(* IEC 61131-3 sources: Multi-PLC-Water-Treatment-Testbed/, 3 files *)

(* ---- plc1_intake.st ---- *)
(* =========================================================================
   PLC1 - INTAKE
   Multi-PLC Water Treatment Testbed
   ---------------------------------------------------------------------------
   Raw-water source intake. Controls the intake pump that fills the treatment
   feed tank, with self-contained process simulation.

   OpenPLC / MatIEC gotchas encoded below:
     1. Located vars (AT %...) and non-located helpers MUST be in SEPARATE
        VAR blocks, else "invalid located variable declaration".
     2. OpenPLC IGNORES initial values on located vars (I/O memory is zeroed
        at start-up). Initialise them in the body on the first scan instead,
        gated by a NON-located first_scan flag (non-located inits ARE honoured).

   Modbus: %MWn -> Holding Register n; %QXn -> Coil. See docs/modbus-map.md.
   ========================================================================= *)

PROGRAM prog0
  VAR
    (* --- Located variables (Modbus-exposed) - NO initial values here --- *)
    source_level     AT %MW0  : INT;
    tank_level       AT %MW1  : INT;
    intake_flow      AT %MW2  : INT;
    pump_status      AT %MW3  : INT;
    pump_cmd         AT %QX0.0 : BOOL;
    low_source_alarm AT %QX0.1 : BOOL;
    tank_high_alarm  AT %QX0.2 : BOOL;
  END_VAR

  VAR
    (* --- Non-located helpers (separate block; inits honoured) --- *)
    first_scan : BOOL := TRUE;
    tick       : INT := 0;
  END_VAR

  (* First-scan initialisation - the only reliable way to seed located vars *)
  IF first_scan THEN
    source_level := 800;
    tank_level   := 300;
    pump_cmd     := TRUE;
    first_scan   := FALSE;
  END_IF;

  tick := tick + 1;
  IF tick >= 20 THEN          (* update process model ~1 Hz at 50 ms scan *)
    tick := 0;

    (* Dry-run protection *)
    IF source_level < 50 THEN
      low_source_alarm := TRUE;
    ELSE
      low_source_alarm := FALSE;
    END_IF;

    (* Pump moves water from source to feed tank when commanded and safe *)
    IF pump_cmd AND (source_level >= 50) THEN
      intake_flow := 100;
      pump_status := 1;
      IF source_level > 0 THEN source_level := source_level - 1; END_IF;
      IF tank_level < 1000 THEN tank_level := tank_level + 2; END_IF;
    ELSE
      intake_flow := 0;
      pump_status := 0;
    END_IF;

    (* Feed tank drains downstream *)
    IF tank_level > 0 THEN tank_level := tank_level - 1; END_IF;

    (* Overflow alarm *)
    IF tank_level >= 950 THEN
      tank_high_alarm := TRUE;
    ELSE
      tank_high_alarm := FALSE;
    END_IF;
  END_IF;
END_PROGRAM

CONFIGURATION Config0
  RESOURCE Res0 ON PLC
    TASK task0(INTERVAL := T#50ms, PRIORITY := 0);
    PROGRAM instance0 WITH task0 : prog0;
  END_RESOURCE
END_CONFIGURATION

(* ---- plc2_treatment.st ---- *)
(* =========================================================================
   PLC2 - TREATMENT
   Multi-PLC Water Treatment Testbed
   ---------------------------------------------------------------------------
   Safety-critical stage: chlorine residual dosing and pH correction.
   Headline attack: zeroing chlorine_setpoint drives chlorine to 0 and raises
   unsafe_water_alarm.

   Scaling: chlorine/pH in hundredths (200 = 2.00 mg/L, 700 = pH 7.00).
   Safe chlorine residual >= 0.50 mg/L (value >= 50).

   OpenPLC gotchas: located vs non-located in SEPARATE VAR blocks; located
   initial values are ignored at runtime, so seed them on first scan.
   See docs/modbus-map.md.
   ========================================================================= *)

PROGRAM prog0
  VAR
    (* --- Located variables (Modbus-exposed) - NO initial values here --- *)
    chlorine_level     AT %MW0  : INT;
    chlorine_setpoint  AT %MW1  : INT;
    ph_level           AT %MW2  : INT;
    ph_setpoint        AT %MW3  : INT;
    dosing_status      AT %MW4  : INT;
    dosing_enable      AT %QX0.0 : BOOL;
    unsafe_water_alarm AT %QX0.1 : BOOL;
    ph_excursion_alarm AT %QX0.2 : BOOL;
  END_VAR

  VAR
    first_scan : BOOL := TRUE;
    tick       : INT := 0;
  END_VAR

  IF first_scan THEN
    chlorine_level    := 200;
    chlorine_setpoint := 200;
    ph_level          := 700;
    ph_setpoint       := 700;
    dosing_status     := 1;
    dosing_enable     := TRUE;
    first_scan        := FALSE;
  END_IF;

  tick := tick + 1;
  IF tick >= 20 THEN
    tick := 0;

    (* Chlorine trends toward setpoint while dosing enabled; setpoint 0 -> decay *)
    IF dosing_enable THEN
      dosing_status := 1;
      IF chlorine_level < chlorine_setpoint THEN
        chlorine_level := chlorine_level + 5;
      ELSIF chlorine_level > chlorine_setpoint THEN
        chlorine_level := chlorine_level - 5;
      END_IF;
    ELSE
      dosing_status := 0;
      IF chlorine_level > 0 THEN chlorine_level := chlorine_level - 5; END_IF;
    END_IF;
    IF chlorine_level < 0 THEN chlorine_level := 0; END_IF;

    (* pH correction trends toward setpoint *)
    IF ph_level < ph_setpoint THEN
      ph_level := ph_level + 2;
    ELSIF ph_level > ph_setpoint THEN
      ph_level := ph_level - 2;
    END_IF;

    (* Safety invariants *)
    IF chlorine_level < 50 THEN
      unsafe_water_alarm := TRUE;
    ELSE
      unsafe_water_alarm := FALSE;
    END_IF;

    IF (ph_level < 650) OR (ph_level > 850) THEN
      ph_excursion_alarm := TRUE;
    ELSE
      ph_excursion_alarm := FALSE;
    END_IF;
  END_IF;
END_PROGRAM

CONFIGURATION Config0
  RESOURCE Res0 ON PLC
    TASK task0(INTERVAL := T#50ms, PRIORITY := 0);
    PROGRAM instance0 WITH task0 : prog0;
  END_RESOURCE
END_CONFIGURATION

(* ---- plc3_distribution.st ---- *)
(* =========================================================================
   PLC3 - DISTRIBUTION
   Multi-PLC Water Treatment Testbed
   ---------------------------------------------------------------------------
   Pressure management and supply via two booster pumps with a pressure-relief
   limit. Attacks: (a) pumps forced OFF -> supply failure; (b) pressure_max
   raised -> relief disabled -> overpressure.

   Scaling: pressure in hundredths of bar (800 = 8.00 bar). Safe hard limit
   = 900. Normal relief setpoint = 800.

   OpenPLC gotchas: located vs non-located in SEPARATE VAR blocks; located
   initial values are ignored at runtime, so seed them on first scan.
   See docs/modbus-map.md.
   ========================================================================= *)

PROGRAM prog0
  VAR
    (* --- Located variables (Modbus-exposed) - NO initial values here --- *)
    pressure           AT %MW0  : INT;
    pressure_max       AT %MW1  : INT;
    booster1_status    AT %MW2  : INT;
    booster2_status    AT %MW3  : INT;
    booster1_cmd       AT %QX0.0 : BOOL;
    booster2_cmd       AT %QX0.1 : BOOL;
    overpressure_alarm AT %QX0.2 : BOOL;
    supply_fail_alarm  AT %QX0.3 : BOOL;
  END_VAR

  VAR
    first_scan : BOOL := TRUE;
    pumps_on   : BOOL := FALSE;
    tick       : INT := 0;
  END_VAR

  IF first_scan THEN
    pressure        := 600;
    pressure_max    := 800;
    booster1_status := 1;
    booster2_status := 1;
    booster1_cmd    := TRUE;
    booster2_cmd    := TRUE;
    first_scan      := FALSE;
  END_IF;

  tick := tick + 1;
  IF tick >= 20 THEN
    tick := 0;

    pumps_on := booster1_cmd OR booster2_cmd;

    IF pumps_on THEN
      pressure := pressure + 30;
    ELSE
      pressure := pressure - 30;
    END_IF;

    (* Relief valve vents above the relief setpoint; raising pressure_max
       (attack) disables relief and lets pressure climb past the 900 limit. *)
    IF pressure > pressure_max THEN
      pressure := pressure_max;
    END_IF;
    IF pressure < 0 THEN pressure := 0; END_IF;

    (* Safety invariants *)
    IF pressure > 900 THEN
      overpressure_alarm := TRUE;
    ELSE
      overpressure_alarm := FALSE;
    END_IF;

    IF pressure < 100 THEN
      supply_fail_alarm := TRUE;
    ELSE
      supply_fail_alarm := FALSE;
    END_IF;

    (* Status mirrors *)
    IF booster1_cmd THEN booster1_status := 1; ELSE booster1_status := 0; END_IF;
    IF booster2_cmd THEN booster2_status := 1; ELSE booster2_status := 0; END_IF;
  END_IF;
END_PROGRAM

CONFIGURATION Config0
  RESOURCE Res0 ON PLC
    TASK task0(INTERVAL := T#50ms, PRIORITY := 0);
    PROGRAM instance0 WITH task0 : prog0;
  END_RESOURCE
END_CONFIGURATION
